ABB RobotStudio station: Solution8.rspag

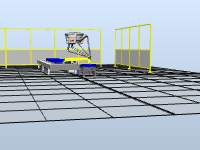
--- station ---
Station Solution8 (saved by RobotStudio 6.8.8307.1040)
Controller System1, task T_ROB1: task frame (RAPID world) sits at (0, 102.45, 1525.12) mm in the station
Controller System1
  mechanical unit ROB_1: IRB360_8_1130_4D_STD_01, 4 joints, base frame (0, 0, 0) mm, rotated rx 180 ry 0 rz 0 deg
Layout (positions relative to the parent item):
  - IRB360_8_1130_4D_STD_01 [mechanism, from Robots\IRB360_8_1130_4D_STD_01.rslib] at (0, 102.45, 1525.12) mm, rotated rx 180 ry 0 rz 0 deg; joint values [0.5605, -0.5879, 1.307, 0] (rad or m)
  - 950_4800_h2 [part, from Equipment\Conveyor 950 4800 h2.rslib]
  - IsoPlate_small_sat [part, from Tools\IsoPlate_small_Binzel.rslib] at (0, -446.74, 631.02) mm, rotated rx 180 ry 0 rz 0 deg
  - Table_small [part] at (719.72, -665.49, -68.21) mm, rotated rx 0 ry 0 rz 92.75 deg
  - SmartComponent_1 [smart component]
      signals: DI move, DO ready
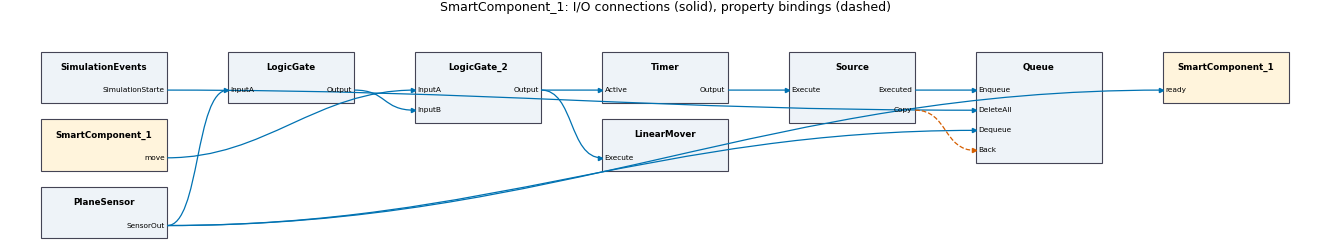
      connections:
        Source.Executed -> Queue.Enqueue
        SimulationEvents.SimulationStarted -> Queue.DeleteAll
        Timer.Output -> Source.Execute
        SmartComponent_1.move -> LogicGate_2.InputA
        LogicGate.Output -> LogicGate_2.InputB
        LogicGate_2.Output -> Timer.Active
        LogicGate_2.Output -> LinearMover.Execute
        PlaneSensor.SensorOut -> Queue.Dequeue
        PlaneSensor.SensorOut -> SmartComponent_1.ready
        PlaneSensor.SensorOut -> LogicGate.InputA
        Source.Copy => Queue.Back
    - Source [smart component, from Components\Source.rslib]
        properties: Source=Cylinder_300_100_2; Copy=Cylinder_300_100_2_102; Parent=(none); Position=[4 0.465743 0.45]; Orientation=[0 0 0]; Transient=false; PhysicsBehavior=0
    - PlaneSensor [smart component, from Components\PlaneSensor.rslib] at (-1255.24, 1389.83, 867.75) mm, rotated rx 180 ry -79.27 rz 180 deg
        properties: Origin=[-0.674457717646954 -1.11176901813793 -1.1568755936615]; Axis1=[0.1 0 0]; Axis2=[0 0.5 0]; SensedPart=(none)
      - _sensorPart_ [part]
    - LinearMover [smart component, from Components\LinearMover.rslib]
        properties: Object=Queue; Direction=[-1 0 0]; Speed=1; Reference=Global; ReferenceObject=(none)
    - LogicGate [smart component, from Components\LogicGate.rslib]
        properties: Operator=NOT; Delay=0
    - Queue [smart component, from Components\Queue.rslib]
        properties: Back=Cylinder_300_100_2_102; Front=Cylinder_300_100_2_99; Queue={26cb5f7c-093d-4500-acf6-86f17ad9141a};{3fc33a52-3250-448e-b337-913ceb35e397};{8442700c-32e3-4c32-83f8-e9cd2cee3a72};{c7e7c410-6e90-4ac1-a3f8-e888f4e302d1}; NumberOfObjects=4
    - SimulationEvents [smart component, from Components\SimulationEvents.rslib]
    - Timer [smart component, from Components\Timer.rslib]
        properties: StartTime=0; Interval=1; Repeat=true; CurrentTime=13.656
    - LogicGate_2 [smart component, from Components\LogicGate.rslib]
        properties: Operator=AND; Delay=0
  - Cylinder_300_100_2 [part, from Training Objects\my_cl.rslib] at (4000, 465.74, 440.04) mm
  - SmartComponent_2 [smart component]
      signals: DI attach
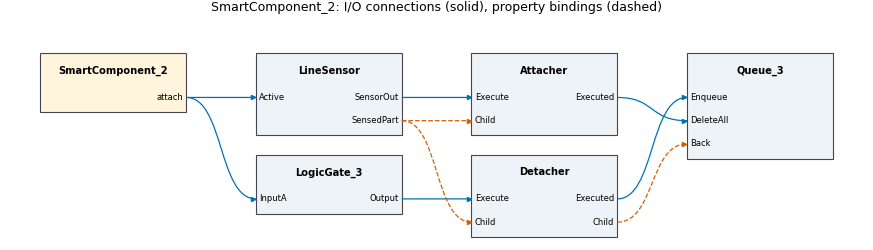
      connections:
        SmartComponent_2.attach -> LineSensor.Active
        LineSensor.SensorOut -> Attacher.Execute
        SmartComponent_2.attach -> LogicGate_3.InputA
        LogicGate_3.Output -> Detacher.Execute
        Detacher.Executed -> Queue_3.Enqueue
        Attacher.Executed -> Queue_3.DeleteAll
        LineSensor.SensedPart => Attacher.Child
        LineSensor.SensedPart => Detacher.Child
        Detacher.Child => Queue_3.Back
    - Attacher [smart component, from Components\Attacher.rslib]
        properties: Parent=IRB360_8_1130_4D_STD_01; Flange=0; Child=Cylinder_300_100_2_98; Mount=false; Offset=[0 0 0]; Orientation=[0 0 0]
    - Detacher [smart component, from Components\Detacher.rslib]
        properties: Child=Cylinder_300_100_2_98; KeepPosition=true
    - LineSensor [smart component, from Components\LineSensor.rslib] at (0, -446.74, 631.02) mm, rotated rx 180 ry 0 rz 0 deg
        properties: Start=[0 0 0.01]; End=[0 0 0.1]; Radius=0; SensedPart=Cylinder_300_100_2_98; SensedPoint=[1.52587890625E-07 -0.446737823486328 0.426347198486328]
      - _sensorPart_ [part]
    - LogicGate_3 [smart component, from Components\LogicGate.rslib]
        properties: Operator=NOT; Delay=0
    - Queue_3 [smart component, from Components\Queue.rslib]
        properties: Back=Cylinder_300_100_2_98; Front=Cylinder_300_100_2_98; Queue={d1b95c8d-deed-4ce4-a727-5991ab0ffbd7}; NumberOfObjects=1
  - Fence_2500 [graphiccomponentgroup, from Equipment\Fence_2500.rslib] at (6026.21, 0, 0) mm
    - Body 1 [part, from Equipment\Fence_2500.rslib]
    - Body 2 [part, from Equipment\Fence_2500.rslib]
  - Fence_2500_3 [graphiccomponentgroup, from Equipment\Fence_2500.rslib] at (6032.55, 2482.69, 0) mm
    - Body 1 [part, from Equipment\Fence_2500.rslib]
    - Body 2 [part, from Equipment\Fence_2500.rslib]
  - Fence_2500_4 [graphiccomponentgroup, from Equipment\Fence_2500.rslib] at (6032.57, -2453.3, 0) mm
    - Body 1 [part, from Equipment\Fence_2500.rslib]
    - Body 2 [part, from Equipment\Fence_2500.rslib]
  - Fence_2500_5 [graphiccomponentgroup, from Equipment\Fence_2500.rslib] at (5926.25, -3232.73, 0) mm, rotated rx 0 ry 0 rz 88.99 deg
    - Body 1 [part, from Equipment\Fence_2500.rslib]
    - Body 2 [part, from Equipment\Fence_2500.rslib]
  - Fence_2500_7 [graphiccomponentgroup, from Equipment\Fence_2500.rslib] at (3445.97, -3191.28, 4.15) mm, rotated rx 0 ry 0 rz 91.05 deg
    - Body 1 [part, from Equipment\Fence_2500.rslib]
    - Body 2 [part, from Equipment\Fence_2500.rslib]
  - Cylinder_300_100_2_98 [part, from Training Objects\my_cl.rslib] at (280, -478.69, 316.37) mm
  - Cylinder_300_100_2_99 [part, from Training Objects\my_cl.rslib] at (352, 465.74, 450) mm
  - Cylinder_300_100_2_100 [part, from Training Objects\my_cl.rslib] at (1360, 465.74, 450) mm
  - Cylinder_300_100_2_101 [part, from Training Objects\my_cl.rslib] at (2344, 465.74, 450) mm
  - Cylinder_300_100_2_102 [part, from Training Objects\my_cl.rslib] at (3352, 465.74, 450) mm
Attachment: IsoPlate_small_sat is attached to IRB360_8_1130_4D_STD_01 / RevoluteLinkPlate
Attachment: LineSensor is attached to IRB360_8_1130_4D_STD_01 / RevoluteLinkPlate
Station logic (signal -> signal, property => property):
  System1.attach0 -> SmartComponent_2.attach
  System1.move0 -> SmartComponent_1.move
  SmartComponent_1.ready -> System1.ready0
Targets, tools, work objects and paths stored in the station and not in the controller backup, written as RAPID:
! task T_ROB1
MODULE Module1
  CONST robtarget Target_10:=[[0,-0.000003553,-960.393260392],[0,1,0,0],[0,0,0,0],[9E+09,9E+09,9E+09,9E+09,9E+09,9E+09]];
ENDMODULE


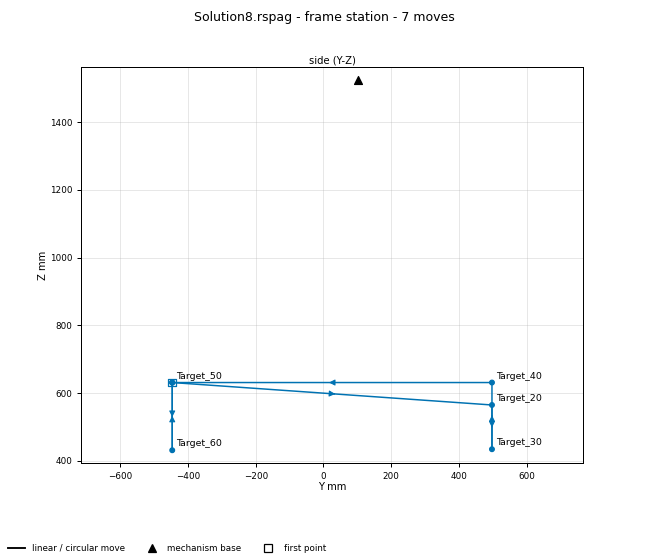
[picture p0: tool path of Solution8.rspag in frame station, 7 of 7 moves have a stored position in this frame; points joined in program order, loops and branches not executed]
--- Backups/System1/RAPID/TASK1/PROGMOD/Module1.mod ---
MODULE Module1
	CONST robtarget Target_20:=[[-0.000044113,395.252359685,-960.393820483],[0,1,0,0],[0,0,0,0],[9E+09,9E+09,9E+09,9E+09,9E+09,9E+09]];
	CONST robtarget Target_30:=[[-0.000146081,395.250433304,-1091.066648557],[0,1,0,0],[0,0,0,0],[9E+09,9E+09,9E+09,9E+09,9E+09,9E+09]];
	CONST robtarget Target_40:=[[-0.000194279,395.249600728,-894.093284384],[0,1,0,0],[0,0,0,0],[9E+09,9E+09,9E+09,9E+09,9E+09,9E+09]];
	CONST robtarget Target_50:=[[-0.000320807,-549.184156874,-894.094290243],[0,1,0,0],[0,0,0,0],[9E+09,9E+09,9E+09,9E+09,9E+09,9E+09]];
	CONST robtarget Target_60:=[[0,-549.183,-1094.095],[0,1,0,0],[0,0,0,0],[9E+09,9E+09,9E+09,9E+09,9E+09,9E+09]];
    !***********************************************************
    !
    ! Module:  Module1
    !
    ! Description:
    !   <Insert description here>
    !
    ! Author: admin
    !
    ! Version: 1.0
    !
    !***********************************************************


    !***********************************************************
    !
    ! Procedure main
    !
    !   This is the entry point of your program
    !
    !***********************************************************
    PROC main()
        SetDO move0, 1;
        WHILE 2+2=4 DO
        Path_10;
        ENDWHILE
    ENDPROC
	PROC Path_10()
	    MoveL Target_50,v1000,z100,tool0\WObj:=wobj0;
        WaitDI ready0, 1;
	    MoveL Target_20,v1000,z100,tool0\WObj:=wobj0;
        WaitRob\InPos;
        SetDO attach0, 1;
	    MoveL Target_30,v1000,z100,tool0\WObj:=wobj0;
	    MoveL Target_40,v1000,z100,tool0\WObj:=wobj0;
	    MoveL Target_50,v1000,z100,tool0\WObj:=wobj0;
	    MoveL Target_60,v1000,z100,tool0\WObj:=wobj0;
        WaitRob\InPos;
        SetDO attach0, 0;
	    MoveL Target_50,v1000,z100,tool0\WObj:=wobj0;
	ENDPROC
	PROC Path_20()

	ENDPROC
ENDMODULE

--- Backups/System1/SYSPAR/EIO.cfg ---
EIO:CFG_1.0:6:1::
#
EIO_SIGNAL:

      -Name "move0" -SignalType "DO" -Access "All"

      -Name "attach0" -SignalType "DO" -Access "All"

      -Name "ready0" -SignalType "DI" -Access "All"
